Staubli VAL3: USERPAGE.pjx

--- USERPAGE.pjx ---
Parameters version=s7.1 stackSize=5000 millimeterUnit=true
Program file=_decode.pgx
Program file=_str2Array.pgx
Program file=clear.pgx
Program file=displayMenu.pgx
Program file=DisplayPt.pgx
Program file=fhmns.pgx
Program file=GetFKey.pgx
Program file=getView.pgx
Program file=hmns.pgx
Program file=isListEmpty.pgx
Program file=leftPos.pgx
Program file=listadd.pgx
Program file=listcreate.pgx
Program file=listcursor.pgx
Program file=listdel.pgx
Program file=listempty.pgx
Program file=listevent.pgx
Program file=listframe.pgx
Program file=listins.pgx
Program file=listredraw.pgx
Program file=listSetSize.pgx
Program file=listupdate.pgx
Program file=midPos.pgx
Program file=msgBox.pgx
Program file=msgBoxDisplay.pgx
Program file=nullKey.pgx
Program file=printScroll.pgx
Program file=read.pgx
Program file=rightPos.pgx
Program file=selectNewField.pgx
Program file=setString.pgx
Program file=setView.pgx
Program file=start.pgx
Program file=stop.pgx
Program file=strAlign.pgx
Program file=strfill.pgx
Program file=strfillchr.pgx
Program file=strlength.pgx
Program file=txtBoxDyn.pgx
Program file=txtBoxDynUpdate.pgx
Program file=type.pgx
Program file=typeBool.pgx
Program file=typeCenter.pgx
Program file=typeDio.pgx
Program file=typeLen.pgx
Program file=typeMenu.pgx
Data file=userPage.dtx

--- USERPAGE.dtx ---
num keyBoard = 277
public num last = 6
public num nBottomX[2] = 12
num nDelimiterCount
public num nFirst = 2
public num nListHeight[2] = 5
public num nTopX[2] = 20
public num nTopY[2] = 1
num nTxtBoxCol
num nTxtBoxRow
num nTxtBoxWidth
public num nView = 4
num posScroll
public num select = -1
num tpsScroll = 103.137
public string alarm
public string background
public string message
public string nameProject = "false"
public string sItems
public string sTitle = "ItemList"
string sWrkString
public string warning
public bool Show
bool bReadWrite = true
bool bUseEscape
bool bUseRefresh
public bool escape
public bool finish
public bool halt
bool readStr
public bool run

--- hmns.pgx ---
public program hmns(num x_nSec, num& x_nHour[], num& x_nMinute[], num& x_nSecond[])
begin
  //-----------------------------------------------------------------------
  //Header begin
  //Description of program
  //  Decompose num seconds in num Hours,minutes, seconds.
  //
  //Input parameters
  //  num x_nSec :
  //    role : put a numerical expression that you want to convert in Hmns
  //
  //Output parameters
  //  num x_nHour :
  //    role : numerical expression that contains Hours
  //  num x_nMinute :
  //    role : numerical expression that contains Minutes
  //  num x_nSecond :
  //    role : numerical expression that contains Seconds
  //
  //Example
  //  call hmns(54200,l_nHour,l_nMinute,l_nSecond)
  //
  //History
  //  Creation : 28-04-08 - f.Rob
  //Header end
  //-----------------------------------------------------------------------
  x_nHour=roundDown(x_nSec/3600)
  x_nMinute=roundDown((x_nSec%3600)/60)
  x_nSecond=roundDown(x_nSec-x_nHour*3600-x_nMinute*60)
end

--- listcreate.pgx ---
public program listCreate(string x_sTitle)
begin
  //-----------------------------------------------------------------------
  //Header begin
  //Description of program
  //  Create a list of data, displays the title x_sTitle,and draw
  //  the list from nTopX and nTopY position of the userPage (),
  //  of nBottomX length and height nListHeight.
  //
  //Input parameters
  //  string x_Title :
  //    role : Title that you want for the list of data
  //
  //Example
  //  Before using listCreate you can use setSizeList for defines all the
  //  parameters of position and size of the menu.
  //  call setSizeList(20,0,18,11)
  //  call listCreate("UserPage")
  //
  //History
  //  Creation : 28-04-08 - f.Rob
  //Header end
  //-----------------------------------------------------------------------
  sTitle=x_sTitle
  //Creation list of data
  call listFrame(sTitle,nTopX,nTopY,nBottomX,nListHeight)
  call listEmpty()
end

--- listins.pgx ---
public program listIns(string& x_sItems[], num x_nPos)
  local num i
  local num l_nSize
begin
  //-----------------------------------------------------------------------
  //Header begin
  //Description of program
  //  Insert an element x_sItem before the number x_nPos.
  //
  //Input parameters
  //  num x_nPos :
  //    role : Position in the array sItems where you want to insert an new Item
  //Output parameters
  //  string x_sItem :
  //    role : Item that you want to insert
  //
  //Example
  //  call listIns("Staubli",3)
  //
  //History
  //  Creation : 28-04-08 - f.Rob
  //Header end
  //-----------------------------------------------------------------------
  l_nSize=size(sItems)-1
  //Test if the position x_nPos is in the array
  if ((x_nPos>=0) and (x_nPos<=l_nSize))
    for i=0 to (size(x_sItems)-1)
      if size(sItems)!=1 or sItems!=""
        //Insert an element in sItems[]
        insert(sItems[x_nPos+i])
        insert(bReadWrite[x_nPos+i])
      endIf
      sItems[x_nPos+i]=x_sItems[i]
      //For default the RW is true
      bReadWrite[x_nPos+i]=true
    endFor
  else
    //Position not in the array
    //Insert the element
    call listAdd(x_sItems)
  endIf
end

--- MIDPOS.pgx ---
public program midPos(string x_sItem, num x_nLength, num x_nPos, string& x_sResult[])
  local string l_sLeft
begin
  //-----------------------------------------------------------------------
  //Header begin
  //Description of program
  //  This program allows to keep x_nLength characters of a string from
  //  a position x_nPos.
  //  The characters before and after x_nPos and x_nPos+x_nLength will be
  //  truncated.
  //
  //Input parameters
  //  string x_sItem :
  //    role : string that you wan to cut
  //  num x_nLength :
  //    role : Length of the characters that you want to keep
  //  num x_nPos :
  //    role : Position to start keeping characters
  //
  //Output parameters
  //  string x_sResult :
  //    role : string truncated
  //
  //Example
  //  call midPos("Staubli Robotics",4,2,sResult)
  //  put(sResult) //Displays "aubl"
  //
  //History
  //  Creation : 28-04-08 - f.Rob
  //Header end
  //-----------------------------------------------------------------------
  // LEFT SIDE
  call leftPos(x_sItem,x_nLength+x_nPos,l_sLeft)
  // update
  x_sResult=l_sLeft
  // RIGHT SIDE
  call rightPos(l_sLeft,x_nLength,x_sResult)
  // OK ....
end
